{attribute 'qualified_only'}
VAR_GLOBAL
	// Filter constants
	fPressureFilterNum 		: LREAL := 0.003137;
	fPressureFilterDenz 	: LREAL := 1.0;
	fPressureFilterDen 		: LREAL := -0.9969;
	fPressureFilterInit 	: LREAL := 0.0;
	
	fPosFilterNum 			: LREAL := 0.003137;
	fPosFilterDenz 			: LREAL := 1.0;
	fPosFilterDen 			: LREAL := -0.9969;
	fPosFilterInit 			: LREAL := 0.0;
	
	fSignalFilterNum 		: LREAL := 0.09516;
	fSignalFilterDenz 		: LREAL := 1.0;
	fSignalFilterDen 		: LREAL := -0.9048;
	fSignalFilterInit 		: LREAL := 0.0;
	
	fDerivatorFilterNum 	: LREAL := 0.0009995;
	fDerivatorFilterDenz 	: LREAL := 1.0;
	fDerivatorFilterDen 	: LREAL := -0.999;
	fDerivatorFilterInit 	: LREAL := 0.0;	
	
	fCutoffFreq             : LREAL := 0.1;
    fDamping                : LREAL := 0.707106781186547;
	fSampleTime             : LREAL := 0.005;
END_VAR

(* stored: Version 1.1.0.1
   GVL G_FilterConstants: Id {454462db-4b24-447f-863f-1528ec74c2bc} *)
